// TIA Portal V20 export
FUNCTION_BLOCK "Pallet_Transport"   // FB14, LAD
{ S7_Optimized_Access := 'TRUE' }
// stored: MemoryReserve 100, SetENOAutomatically false
   VAR_INPUT
      Source_X : SInt;
      Source_Z : SInt;
      Destination_X : SInt;
      Destination_Z : SInt;
      Stations : Array[0..3] of "Station";
      Station_ST31 : "Station";
      Station_ST32 : "Station";
      Station_ST34 : "Station";
      Station_Lift : "Station";
      Lift_On_The_Floor : Bool;
      Lift_On_Num_Floor : SInt;
      Manual : Bool;
   END_VAR
   VAR_OUTPUT
      oButton_StS_StD_LED : Bool;
      oStatus_HMI_StS_StD : Bool;
      oStatus_HMI_StD_StS : Bool;
      oCentering : Bool;
      Stop_Drive_Button : Bool;
      Stop_Drive_HMI : Bool;
   END_VAR
   VAR_IN_OUT
      iDriveST31_Param : "SEW_MOVIKIT_VelocityDrive_SETPOINTS_V2.1";
      oDriveST31_Param : "SEW_MOVIKIT_VelocityDrive_STATUS_V2.1";
      iDriveST32_Param : "SEW_MOVIKIT_VelocityDrive_SETPOINTS_V2.1";
      oDriveST32_Param : "SEW_MOVIKIT_VelocityDrive_STATUS_V2.1";
      iDriveST34_Param : "SEW_MOVIKIT_VelocityDrive_SETPOINTS_V2.1";
      oDriveST34_Param : "SEW_MOVIKIT_VelocityDrive_STATUS_V2.1";
      iDriveLift_Param : "SEW_MOVIKIT_VelocityDrive_SETPOINTS_V2.1";
      oDriveLiftParam : "SEW_MOVIKIT_VelocityDrive_STATUS_V2.1";
      HMI_StS_StD : Bool;
      HMI_StD_StS : Bool;
   END_VAR
   VAR
      Drive_To_Destination : Bool;
      Set_Speed : Int;
      Set_Speed_Reverse : Int;
      CommunicationOk : Bool;
      Jog_StS : Bool;
      Jog_StD : Bool;
      CenteringStep : Int;
      TON_Centering : TON_TIME;
      trigTimeout { S7_SetPoint := 'True'} : R_TRIG;
      Trig_StS_StD { S7_SetPoint := 'True'} : Bool;
      Trig_StD_StS : Bool;
      Reset_StS_StD : Bool;
      Reset_StD_StS : Bool;
      Timer_Drive_Error_Button : TON_TIME;
      Timer_Drive_Error_HMI : TON_TIME;
      STOP_DRIVERS { S7_SetPoint := 'True'} : Bool;
      PathFree : Bool;
   END_VAR
   VAR_TEMP
      LED_StD_STS : Bool;
      LED_StS_STD : Bool;
      minIdx : SInt;
      maxIdx : SInt;
      i : SInt;
   END_VAR
   VAR CONSTANT
      ACC : Int := 300;
      DCC : Int := 400;
      SPEED_BACK : Int := -100;
      SPEED_FWD : Int := 100;
   END_VAR
   VAR_TEMP   // added for the SCL form of the ladder/FBD networks
      _w1 : Bool;
      _w2 : Bool;
      _w3 : Bool;
      _w4 : Bool;
   END_VAR
BEGIN

REGION Network 1: Reset commands
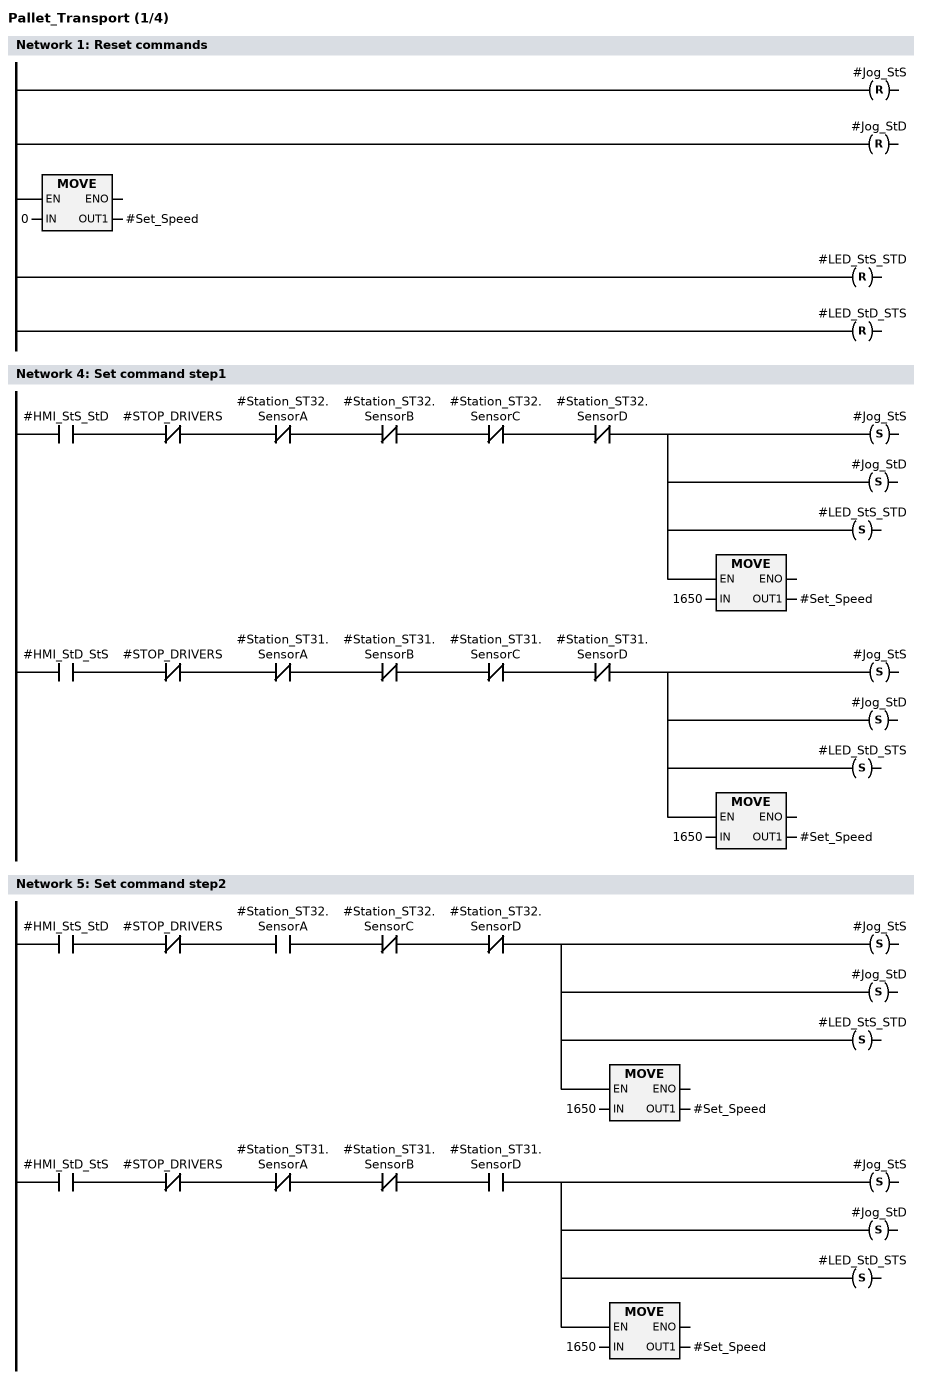
   RUNG wire#powerrail
      R_Coil( #Jog_StS )
   END_RUNG
   RUNG wire#powerrail
      R_Coil( #Jog_StD )
   END_RUNG
   RUNG wire#powerrail
      Move(in := 0, out1 => #Set_Speed)
   END_RUNG
   RUNG wire#powerrail
      R_Coil( #LED_StS_STD )
   END_RUNG
   RUNG wire#powerrail
      R_Coil( #LED_StD_STS )
   END_RUNG
   // the same network as SCL:
   #Jog_StS := FALSE;
   #Jog_StD := FALSE;
   #Set_Speed := 0;
   #LED_StS_STD := FALSE;
   #LED_StD_STS := FALSE;
END_REGION

REGION Network 2 (SCL): Triggers STOP_DRIVERS after 8 s of active move command without motion
   #Timer_Drive_Error_HMI(
                          IN :=
                          (
                          #HMI_StS_StD OR
                          #HMI_StD_StS
                          )
                          AND NOT (
                          #oDriveST31_Param.x_Bit_4_Motor_turning OR
                          #oDriveST32_Param.x_Bit_4_Motor_turning
                          ),
                          PT := T#10s
   );

   IF #Timer_Drive_Error_Button.Q THEN
       #STOP_DRIVERS := TRUE;
       #Stop_Drive_Button := TRUE;
   END_IF;

   IF #Timer_Drive_Error_HMI.Q THEN
       #STOP_DRIVERS := TRUE;
       #Stop_Drive_HMI := TRUE;
       #HMI_StS_StD := FALSE;
       #HMI_StD_StS := FALSE;
   END_IF;

   IF "HMI".Reset_Motors THEN
       #STOP_DRIVERS := FALSE;
       #Stop_Drive_Button := FALSE;
       #Stop_Drive_HMI := FALSE;
   END_IF;
END_REGION

REGION Network 3 (SCL): Check free path
   #minIdx := MIN_SINT(IN1:=#Source_X, IN2:=#Destination_X);

   #maxIdx := MAX_SINT(IN1:=#Source_X, IN2:=#Destination_X);

   #PathFree := TRUE;

   FOR #i := #minIdx + 1 TO #maxIdx DO
       IF #Stations[#i].isEmpty = FALSE THEN
           #PathFree := FALSE;
           EXIT;
       END_IF;
   END_FOR;
END_REGION

REGION Network 4: Set command step1
   RUNG wire#powerrail
      Contact( #HMI_StS_StD )
      I_Contact( #STOP_DRIVERS )
      I_Contact( #Station_ST32.SensorA )
      I_Contact( #Station_ST32.SensorB )
      I_Contact( #Station_ST32.SensorC )
      I_Contact( #Station_ST32.SensorD )
      wire#w1
      S_Coil( #Jog_StS )
   END_RUNG
   RUNG wire#w1
      S_Coil( #Jog_StD )
   END_RUNG
   RUNG wire#w1
      S_Coil( #LED_StS_STD )
   END_RUNG
   RUNG wire#w1
      Move(in := 1650, out1 => #Set_Speed)
   END_RUNG
   RUNG wire#powerrail
      Contact( #HMI_StD_StS )
      I_Contact( #STOP_DRIVERS )
      I_Contact( #Station_ST31.SensorA )
      I_Contact( #Station_ST31.SensorB )
      I_Contact( #Station_ST31.SensorC )
      I_Contact( #Station_ST31.SensorD )
      wire#w2
      S_Coil( #Jog_StS )
   END_RUNG
   RUNG wire#w2
      S_Coil( #Jog_StD )
   END_RUNG
   RUNG wire#w2
      S_Coil( #LED_StD_STS )
   END_RUNG
   RUNG wire#w2
      Move(in := 1650, out1 => #Set_Speed)
   END_RUNG
   // the same network as SCL:
   IF #HMI_StS_StD AND NOT #STOP_DRIVERS AND NOT #Station_ST32.SensorA AND NOT #Station_ST32.SensorB AND NOT #Station_ST32.SensorC AND NOT #Station_ST32.SensorD THEN
       #Jog_StS := TRUE;
       #Jog_StD := TRUE;
       #LED_StS_STD := TRUE;
       #Set_Speed := 1650;
   END_IF;
   IF #HMI_StD_StS AND NOT #STOP_DRIVERS AND NOT #Station_ST31.SensorA AND NOT #Station_ST31.SensorB AND NOT #Station_ST31.SensorC AND NOT #Station_ST31.SensorD THEN
       #Jog_StS := TRUE;
       #Jog_StD := TRUE;
       #LED_StD_STS := TRUE;
       #Set_Speed := 1650;
   END_IF;
END_REGION

REGION Network 5: Set command step2
   RUNG wire#powerrail
      Contact( #HMI_StS_StD )
      I_Contact( #STOP_DRIVERS )
      Contact( #Station_ST32.SensorA )
      I_Contact( #Station_ST32.SensorC )
      I_Contact( #Station_ST32.SensorD )
      wire#w1
      S_Coil( #Jog_StS )
   END_RUNG
   RUNG wire#w1
      S_Coil( #Jog_StD )
   END_RUNG
   RUNG wire#w1
      S_Coil( #LED_StS_STD )
   END_RUNG
   RUNG wire#w1
      Move(in := 1650, out1 => #Set_Speed)
   END_RUNG
   RUNG wire#powerrail
      Contact( #HMI_StD_StS )
      I_Contact( #STOP_DRIVERS )
      I_Contact( #Station_ST31.SensorA )
      I_Contact( #Station_ST31.SensorB )
      Contact( #Station_ST31.SensorD )
      wire#w2
      S_Coil( #Jog_StS )
   END_RUNG
   RUNG wire#w2
      S_Coil( #Jog_StD )
   END_RUNG
   RUNG wire#w2
      S_Coil( #LED_StD_STS )
   END_RUNG
   RUNG wire#w2
      Move(in := 1650, out1 => #Set_Speed)
   END_RUNG
   // the same network as SCL:
   IF #HMI_StS_StD AND NOT #STOP_DRIVERS AND #Station_ST32.SensorA AND NOT #Station_ST32.SensorC AND NOT #Station_ST32.SensorD THEN
       #Jog_StS := TRUE;
       #Jog_StD := TRUE;
       #LED_StS_STD := TRUE;
       #Set_Speed := 1650;
   END_IF;
   IF #HMI_StD_StS AND NOT #STOP_DRIVERS AND NOT #Station_ST31.SensorA AND NOT #Station_ST31.SensorB AND #Station_ST31.SensorD THEN
       #Jog_StS := TRUE;
       #Jog_StD := TRUE;
       #LED_StD_STS := TRUE;
       #Set_Speed := 1650;
   END_IF;
END_REGION

REGION Network 6: Set command step3
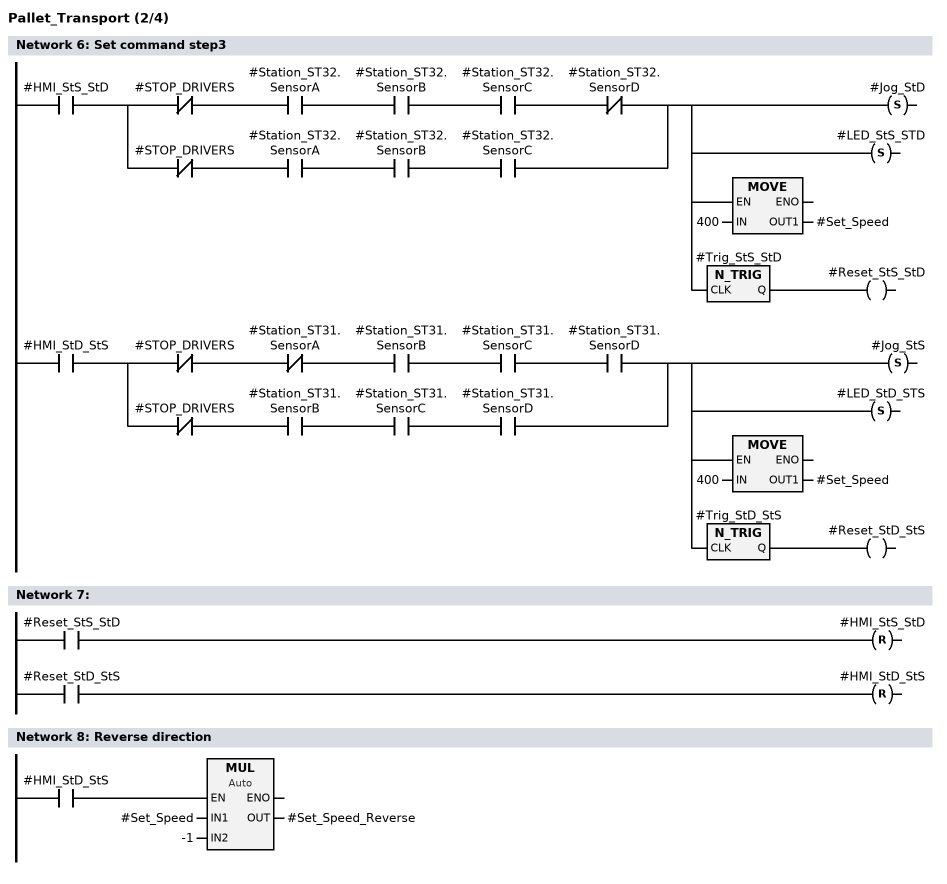
   RUNG wire#powerrail
      Contact( #HMI_StS_StD )
      wire#w1
      I_Contact( #STOP_DRIVERS )
      Contact( #Station_ST32.SensorA )
      Contact( #Station_ST32.SensorB )
      Contact( #Station_ST32.SensorC )
      I_Contact( #Station_ST32.SensorD )
      wire#w2
      S_Coil( #Jog_StD )
   END_RUNG
   RUNG wire#w1
      I_Contact( #STOP_DRIVERS )
      Contact( #Station_ST32.SensorA )
      Contact( #Station_ST32.SensorB )
      Contact( #Station_ST32.SensorC )
   END_RUNG wire#w2
   RUNG wire#w2
      S_Coil( #LED_StS_STD )
   END_RUNG
   RUNG wire#w2
      Move(in := 400, out1 => #Set_Speed)
   END_RUNG
   RUNG wire#w2
      N_Trig( #Trig_StS_StD )
      Coil( #Reset_StS_StD )
   END_RUNG
   RUNG wire#powerrail
      Contact( #HMI_StD_StS )
      wire#w3
      I_Contact( #STOP_DRIVERS )
      I_Contact( #Station_ST31.SensorA )
      Contact( #Station_ST31.SensorB )
      Contact( #Station_ST31.SensorC )
      Contact( #Station_ST31.SensorD )
      wire#w4
      S_Coil( #Jog_StS )
   END_RUNG
   RUNG wire#w3
      I_Contact( #STOP_DRIVERS )
      Contact( #Station_ST31.SensorB )
      Contact( #Station_ST31.SensorC )
      Contact( #Station_ST31.SensorD )
   END_RUNG wire#w4
   RUNG wire#w4
      S_Coil( #LED_StD_STS )
   END_RUNG
   RUNG wire#w4
      Move(in := 400, out1 => #Set_Speed)
   END_RUNG
   RUNG wire#w4
      N_Trig( #Trig_StD_StS )
      Coil( #Reset_StD_StS )
   END_RUNG
   // the same network as SCL:
   #_w1 := #HMI_StS_StD AND ((NOT #STOP_DRIVERS AND #Station_ST32.SensorA AND #Station_ST32.SensorB AND #Station_ST32.SensorC AND NOT #Station_ST32.SensorD) OR (NOT #STOP_DRIVERS AND #Station_ST32.SensorA AND #Station_ST32.SensorB AND #Station_ST32.SensorC));
   IF #_w1 THEN
       #Jog_StD := TRUE;
       #LED_StS_STD := TRUE;
       #Set_Speed := 400;
   END_IF;
   #_w2 := NOT #_w1 AND #Trig_StS_StD;   // falling edge
   #Trig_StS_StD := #_w1;
   #Reset_StS_StD := #_w2;
   #_w3 := #HMI_StD_StS AND ((NOT #STOP_DRIVERS AND NOT #Station_ST31.SensorA AND #Station_ST31.SensorB AND #Station_ST31.SensorC AND #Station_ST31.SensorD) OR (NOT #STOP_DRIVERS AND #Station_ST31.SensorB AND #Station_ST31.SensorC AND #Station_ST31.SensorD));
   IF #_w3 THEN
       #Jog_StS := TRUE;
       #LED_StD_STS := TRUE;
       #Set_Speed := 400;
   END_IF;
   #_w4 := NOT #_w3 AND #Trig_StD_StS;   // falling edge
   #Trig_StD_StS := #_w3;
   #Reset_StD_StS := #_w4;
END_REGION

REGION Network 7
   RUNG wire#powerrail
      Contact( #Reset_StS_StD )
      R_Coil( #HMI_StS_StD )
   END_RUNG
   RUNG wire#powerrail
      Contact( #Reset_StD_StS )
      R_Coil( #HMI_StD_StS )
   END_RUNG
   // the same network as SCL:
   IF #Reset_StS_StD THEN #HMI_StS_StD := FALSE; END_IF;
   IF #Reset_StD_StS THEN #HMI_StD_StS := FALSE; END_IF;
END_REGION

REGION Network 8: Reverse direction
   RUNG wire#powerrail
      Contact( #HMI_StD_StS )
      Mul(in1 := #Set_Speed, in2 := -1, out => #Set_Speed_Reverse)
   END_RUNG
   // the same network as SCL:
   IF #HMI_StD_StS THEN #Set_Speed_Reverse := #Set_Speed * (-1); END_IF;
END_REGION

REGION Network 9: StS Drive
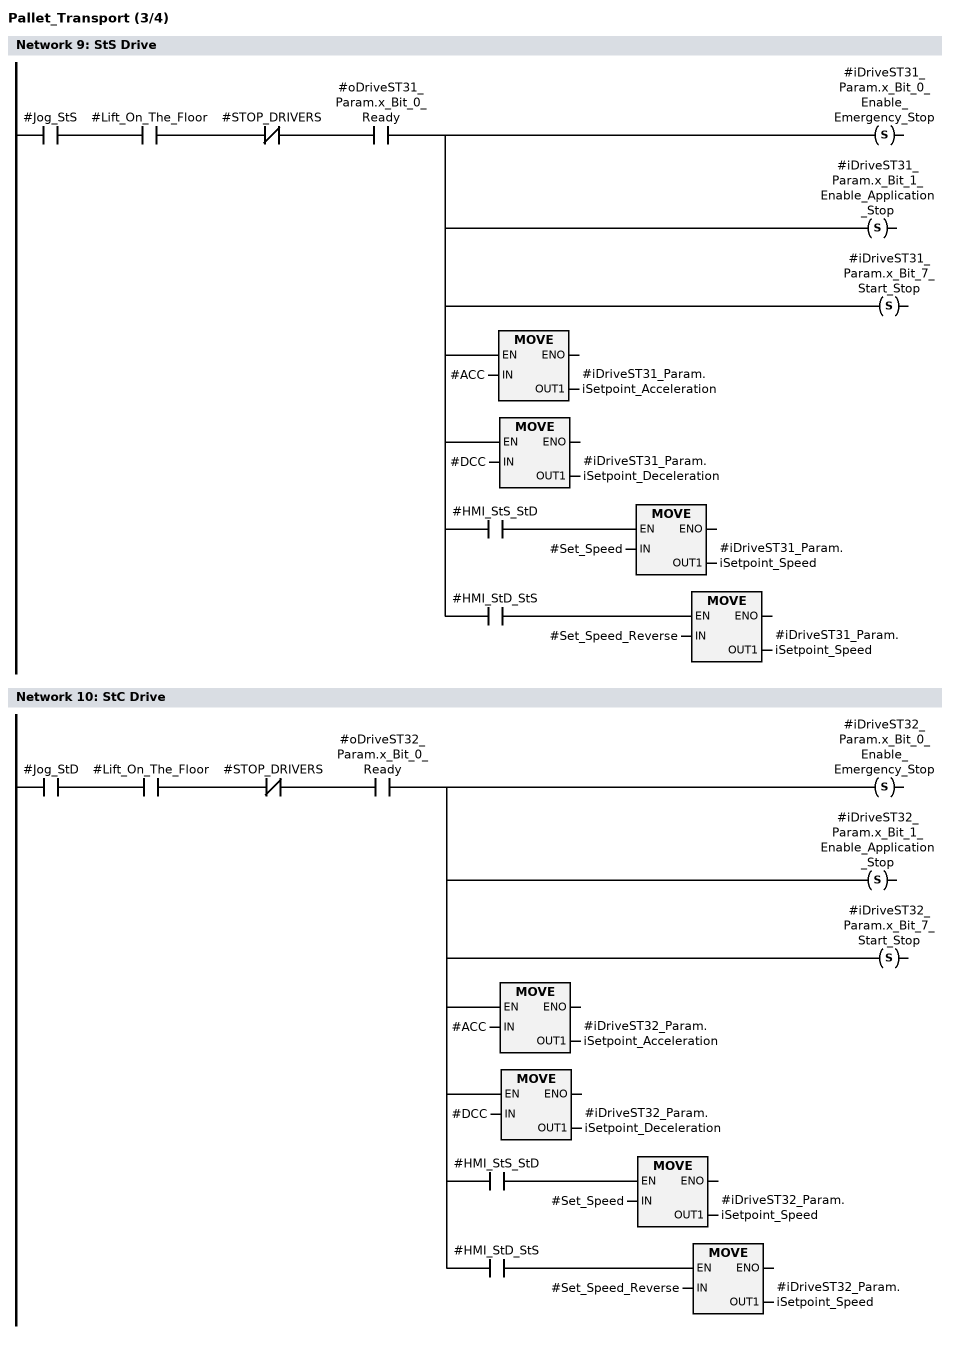
   RUNG wire#powerrail
      Contact( #Jog_StS )
      Contact( #Lift_On_The_Floor )
      I_Contact( #STOP_DRIVERS )
      Contact( #oDriveST31_Param.x_Bit_0_Ready )
      wire#w1
      S_Coil( #iDriveST31_Param.x_Bit_0_Enable_Emergency_Stop )
   END_RUNG
   RUNG wire#w1
      S_Coil( #iDriveST31_Param.x_Bit_1_Enable_Application_Stop )
   END_RUNG
   RUNG wire#w1
      S_Coil( #iDriveST31_Param.x_Bit_7_Start_Stop )
   END_RUNG
   RUNG wire#w1
      Move(in := #ACC, out1 => #iDriveST31_Param.iSetpoint_Acceleration)
   END_RUNG
   RUNG wire#w1
      Move(in := #DCC, out1 => #iDriveST31_Param.iSetpoint_Deceleration)
   END_RUNG
   RUNG wire#w1
      Contact( #HMI_StS_StD )
      Move(in := #Set_Speed, out1 => #iDriveST31_Param.iSetpoint_Speed)
   END_RUNG
   RUNG wire#w1
      Contact( #HMI_StD_StS )
      Move(in := #Set_Speed_Reverse, out1 => #iDriveST31_Param.iSetpoint_Speed)
   END_RUNG
   // the same network as SCL:
   #_w1 := #Jog_StS AND #Lift_On_The_Floor AND NOT #STOP_DRIVERS AND #oDriveST31_Param.x_Bit_0_Ready;
   IF #_w1 THEN
       #iDriveST31_Param.x_Bit_0_Enable_Emergency_Stop := TRUE;
       #iDriveST31_Param.x_Bit_1_Enable_Application_Stop := TRUE;
       #iDriveST31_Param.x_Bit_7_Start_Stop := TRUE;
       #iDriveST31_Param.iSetpoint_Acceleration := #ACC;
       #iDriveST31_Param.iSetpoint_Deceleration := #DCC;
   END_IF;
   IF #_w1 AND #HMI_StS_StD THEN #iDriveST31_Param.iSetpoint_Speed := #Set_Speed; END_IF;
   IF #_w1 AND #HMI_StD_StS THEN #iDriveST31_Param.iSetpoint_Speed := #Set_Speed_Reverse; END_IF;
END_REGION

REGION Network 10: StC Drive
   RUNG wire#powerrail
      Contact( #Jog_StD )
      Contact( #Lift_On_The_Floor )
      I_Contact( #STOP_DRIVERS )
      Contact( #oDriveST32_Param.x_Bit_0_Ready )
      wire#w1
      S_Coil( #iDriveST32_Param.x_Bit_0_Enable_Emergency_Stop )
   END_RUNG
   RUNG wire#w1
      S_Coil( #iDriveST32_Param.x_Bit_1_Enable_Application_Stop )
   END_RUNG
   RUNG wire#w1
      S_Coil( #iDriveST32_Param.x_Bit_7_Start_Stop )
   END_RUNG
   RUNG wire#w1
      Move(in := #ACC, out1 => #iDriveST32_Param.iSetpoint_Acceleration)
   END_RUNG
   RUNG wire#w1
      Move(in := #DCC, out1 => #iDriveST32_Param.iSetpoint_Deceleration)
   END_RUNG
   RUNG wire#w1
      Contact( #HMI_StS_StD )
      Move(in := #Set_Speed, out1 => #iDriveST32_Param.iSetpoint_Speed)
   END_RUNG
   RUNG wire#w1
      Contact( #HMI_StD_StS )
      Move(in := #Set_Speed_Reverse, out1 => #iDriveST32_Param.iSetpoint_Speed)
   END_RUNG
   // the same network as SCL:
   #_w1 := #Jog_StD AND #Lift_On_The_Floor AND NOT #STOP_DRIVERS AND #oDriveST32_Param.x_Bit_0_Ready;
   IF #_w1 THEN
       #iDriveST32_Param.x_Bit_0_Enable_Emergency_Stop := TRUE;
       #iDriveST32_Param.x_Bit_1_Enable_Application_Stop := TRUE;
       #iDriveST32_Param.x_Bit_7_Start_Stop := TRUE;
       #iDriveST32_Param.iSetpoint_Acceleration := #ACC;
       #iDriveST32_Param.iSetpoint_Deceleration := #DCC;
   END_IF;
   IF #_w1 AND #HMI_StS_StD THEN #iDriveST32_Param.iSetpoint_Speed := #Set_Speed; END_IF;
   IF #_w1 AND #HMI_StD_StS THEN #iDriveST32_Param.iSetpoint_Speed := #Set_Speed_Reverse; END_IF;
END_REGION

REGION Network 11: StS -> StD Status
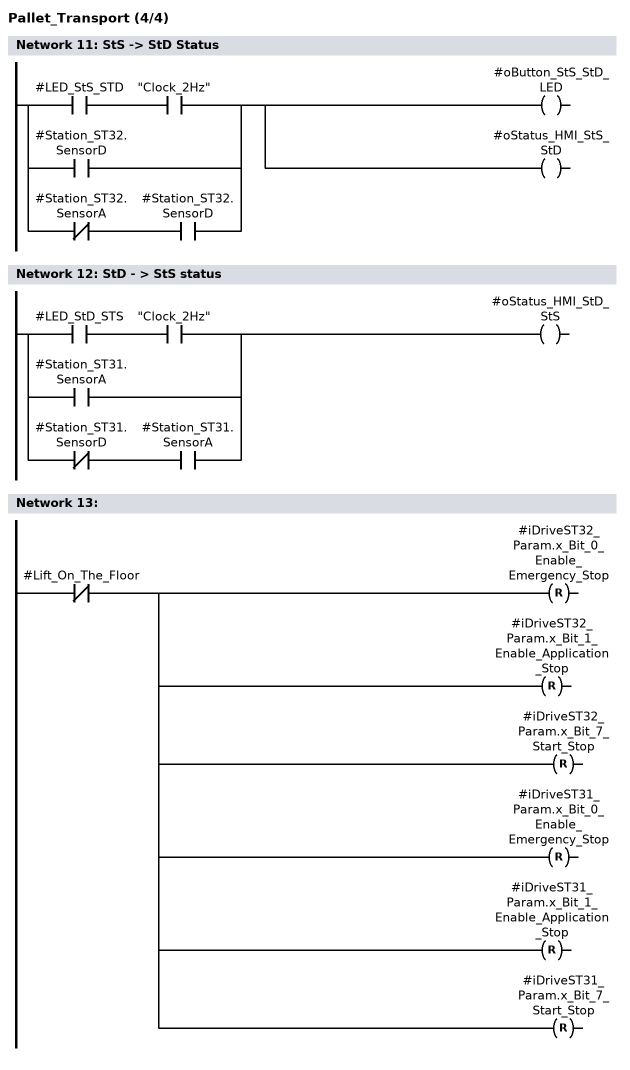
   RUNG wire#powerrail
      Contact( #LED_StS_STD )
      Contact( "Clock_2Hz" )
      wire#w1
      Coil( #oButton_StS_StD_LED )
   END_RUNG
   RUNG wire#powerrail
      Contact( #Station_ST32.SensorD )
   END_RUNG wire#w1
   RUNG wire#powerrail
      I_Contact( #Station_ST32.SensorA )
      Contact( #Station_ST32.SensorD )
   END_RUNG wire#w1
   RUNG wire#w1
      Coil( #oStatus_HMI_StS_StD )
   END_RUNG
   // the same network as SCL:
   #oButton_StS_StD_LED := (#LED_StS_STD AND "Clock_2Hz") OR #Station_ST32.SensorD OR (NOT #Station_ST32.SensorA AND #Station_ST32.SensorD);
   #oStatus_HMI_StS_StD := #oButton_StS_StD_LED;
END_REGION

REGION Network 12: StD - > StS status
   RUNG wire#powerrail
      Contact( #LED_StD_STS )
      Contact( "Clock_2Hz" )
      wire#w1
      Coil( #oStatus_HMI_StD_StS )
   END_RUNG
   RUNG wire#powerrail
      Contact( #Station_ST31.SensorA )
   END_RUNG wire#w1
   RUNG wire#powerrail
      I_Contact( #Station_ST31.SensorD )
      Contact( #Station_ST31.SensorA )
   END_RUNG wire#w1
   // the same network as SCL:
   #oStatus_HMI_StD_StS := (#LED_StD_STS AND "Clock_2Hz") OR #Station_ST31.SensorA OR (NOT #Station_ST31.SensorD AND #Station_ST31.SensorA);
END_REGION

REGION Network 13
   RUNG wire#powerrail
      I_Contact( #Lift_On_The_Floor )
      wire#w1
      R_Coil( #iDriveST32_Param.x_Bit_0_Enable_Emergency_Stop )
   END_RUNG
   RUNG wire#w1
      R_Coil( #iDriveST32_Param.x_Bit_1_Enable_Application_Stop )
   END_RUNG
   RUNG wire#w1
      R_Coil( #iDriveST32_Param.x_Bit_7_Start_Stop )
   END_RUNG
   RUNG wire#w1
      R_Coil( #iDriveST31_Param.x_Bit_0_Enable_Emergency_Stop )
   END_RUNG
   RUNG wire#w1
      R_Coil( #iDriveST31_Param.x_Bit_1_Enable_Application_Stop )
   END_RUNG
   RUNG wire#w1
      R_Coil( #iDriveST31_Param.x_Bit_7_Start_Stop )
   END_RUNG
   // the same network as SCL:
   IF NOT #Lift_On_The_Floor THEN
       #iDriveST32_Param.x_Bit_0_Enable_Emergency_Stop := FALSE;
       #iDriveST32_Param.x_Bit_1_Enable_Application_Stop := FALSE;
       #iDriveST32_Param.x_Bit_7_Start_Stop := FALSE;
       #iDriveST31_Param.x_Bit_0_Enable_Emergency_Stop := FALSE;
       #iDriveST31_Param.x_Bit_1_Enable_Application_Stop := FALSE;
       #iDriveST31_Param.x_Bit_7_Start_Stop := FALSE;
   END_IF;
END_REGION
END_FUNCTION_BLOCK
